Omron CX-Programmer project NewProject (CX-Programmer 9.03)

# PLC NewPLC1: CP1L L

## Global symbols (name address type ; comment)
0.00 BOOL  ; tombol 1
0.01 BOOL  ; tombol 2
0.02 BOOL  ; tombol MC
1.00 BOOL  ; lampu 1
1.01 BOOL  ; lampu 2
1.02 BOOL  ; buzzer

## Program NewProgram1 (cyclic task 0)
; Acara Lomba
Local symbols
d BOOL

### Section Section1
; sesi tanya jawab

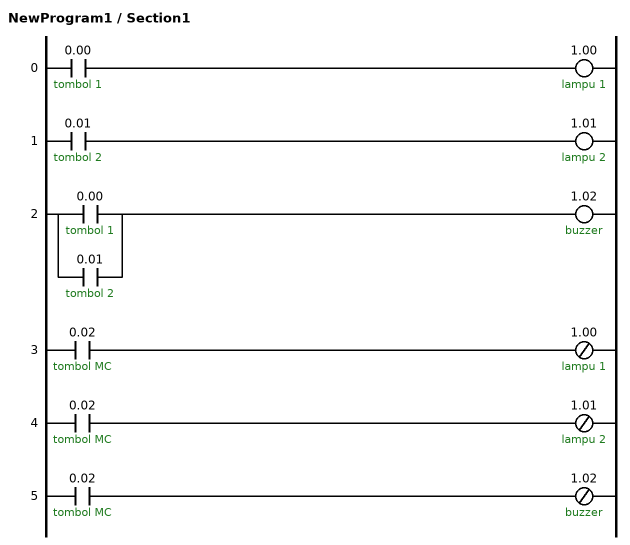
; rung 0
LD 0.00  ; tombol 1
OUT 1.00  ; lampu 1
; rung 1
LD 0.01  ; tombol 2
OUT 1.01  ; lampu 2
; rung 2
LD 0.00  ; tombol 1
OR 0.01  ; tombol 2
OUT 1.02  ; buzzer
; rung 3
LD 0.02  ; tombol MC
OUTNOT 1.00  ; lampu 1
; rung 4
LD 0.02  ; tombol MC
OUTNOT 1.01  ; lampu 2
; rung 5
LD 0.02  ; tombol MC
OUTNOT 1.02  ; buzzer

### Section END
; rung 0
END(001)